FUNCTION_BLOCK Fb2PosControl (* Регулятор двухпозиционный. *)
  (* Standard: 61499-1; Description: Регулятор двухпозиционный. Simple FB with one algorithm *)
  (* Version 2.1, 2026-03-20, VA, LIB_PLC *)
  (* Documentation:
  // Регулятор двухпозиционный. //       Db2PosControl //     +---------------+ //     | Fb2PosControl | //  ->-|PV           OP|->- //    -|SP             | //    -|HYST           | //     +---------------+ // Применение. // // Двухпозиционный регулятор используется как простейший регулятор температуры, давления, уровня. // Условное графическое обозначение. // //      +---------------+ //      |               | //      |    +--<--+--  | //      |    |     |    | // ER->-|    v     ^    |->-OP //      |    |     |    | //      |  --+-->--+    | //      |               | //      +---------------+ // Статическая характеристика. // //                 OP //                  ^ //                  | //           ***<***1***<****** //           *      |      * //           v      |      ^ //           *      |      * // -ER <--******>***0***>***--> +ER //           |      |      | //           |<---->|<---->| //             HYST   HYST // Временная характеристика. // // ^ PV,SP // |         PV // |----------*---------------*------ // |         * *             * *   | // |        *   *           *   *  |  SP + HYST // |       *     *         *       | // |======*=======*=======*========== SP // |     *         *     *         | // |    *           *   *          |  SP - HYST // |   *             * *           | // |--*---------------*-------------- // | *  // |* // +-----------------------------------------> t[s] // // ^ OP // | // 1***********       ********* // |          *       *       * // 0----------*********-------***------------> t[s] // Схема включения. // //                  +---------------+ //                  |               |   Объект управления //                  |    +--<--+--  |     +-----------+ //        +---+ ER  |    |     |    | OP  |     K     | // SP-->--| + |-->--|    v     ^    |-->--| --------- |-->--+-->PV // PV  +--| - |     |    |     |    |     | T * s + 1 |     | //     |  +---+     |  --+-->--+    |     +-----------+     | //     |            |               |                       | //     |            +---------------+                       | //     |                                                    | //     +----------------------------------------------------+
  *)
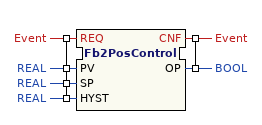
  EVENT_INPUT
    REQ WITH PV, SP, HYST; (* Normal Execution Request *)
  END_EVENT
  EVENT_OUTPUT
    CNF WITH OP; (* Execution Confirmation *)
  END_EVENT
  VAR_INPUT
    PV : REAL := 0.0; (* Измеренное значение регулируемого параметра. *)
    SP : REAL := 0.0; (* Заданное значение регулируемого параметра. *)
    HYST : REAL := 0.0; (* Гистерезис > 0. *)
  END_VAR
  VAR_OUTPUT
    OP : BOOL := FALSE; (* Выход управляющего сигнала. *)
  END_VAR
  VAR
    ER : REAL := 0.0; (* Ошибка регулирования. *)
  END_VAR
  EC_STATES
    REQ : REQ -> CNF;
  END_STATES
  ALGORITHM REQ IN ST:
// Ошибка регулирования.
ER := SP - PV;

// Регулятор двухпозиционный.
IF (ER >= HYST) THEN
	OP := TRUE;
END_IF;

IF (ER <= HYST * (-1.0)) THEN
	OP := FALSE;
END_IF;

// @COPYLEFT ALL WRONGS RESERVED :)
// Author: VA
// Contacts: DIY.PLC.314@gmail.com
// Date start LIB_PLC: 2014
// License: GNU GPL-2.0-or-later
// https://www.gnu.org/licenses/old-licenses/gpl-2.0.html
// https://www.youtube.com/watch?v=n1F_MfLRlX0
// https://www.youtube.com/@DIY_PLC
// https://github.com/DIYPLC/LIB_PLC
// https://oshwlab.com/diy.plc.314/PLC_HW1_SW1
// https://3dtoday.ru/3d-models/mechanical-parts/body/korpus-na-din-reiku
// https://t.me/DIY_PLC
  END_ALGORITHM
END_FUNCTION_BLOCK
